//---------------------------------------------------------------------------------------------------------------
//
//  HAUD 2024.11.21
//
//
//  fb_Instance
//-----------------------------------------------------------------------------
//  - base class for my process instance to work with fb_ProcessCollector
//
//  - _nProcess --> whoami, this is me
//
//  - fb_ProcessCollector[_nProcess].Cycle() is called in APPLICATION(PRG)
//    - handles range of XtsStations
//    - range must be closed and in consecutive order
//
//    - combines states into bitmasks, one bit per XtsStation
//    - controls forwarding of commands to range of XtsStations 
//      (see fb_ProcessCollector.Cycle())
//
//  - reference to all _ItfProcessCollector(I_ProcessCollector)[]
//    - _ItfProcessCollector[nProcess] Get/Set properties and methods
//
//  - Control / State of my process
//    - datafield for control and state provided
//    - _Ctrl 
//      --> commands to my process; fb_ProcessCollector[_nProcess]
//      --> is linked (REF=) automatically in Check()
//
//      Cmd               : E_PROCESS_CTRL; // command enum for my process
//      ProcessTarget     : UINT;           // target of my process
//      ActivateStation   : WORD;           // is checked for every job
//                                          // every bit is a XtsStation
//
//      NestMask          : BYTE;           // one mask for all XtsStations
//      - every bit is a PosStop in a XtsStation
//      - copied to every XtsStation in my process when movers are about to leave
//
//    - _State
//      --> satus information from my process
//      --> check for plausible StationLast / StationFirst range of XtsStations
//
//      State             : E_PROCESS_STATE;  // state enuum from my process
//      Result            : E_PROGRESS;       // substate from my process, BUSY signals state is ready for interaction
//      Check             : E_PROCESS_CHECK;  // plausibility check of StationLast and StationFirst 
//
//
//  - basic check and var names, so you can build your procedures with it
//
//  - processes may be connected via linked list, you decide.
//    - linked list for processes is intended to work as job buffer
//    - linked list provides information via ST_PROCESS_DATA, 
//      add what you have to in there
//    - linked ist to all process instances provided
//
//  - inherit this base class for your application, call Check() cyclic
//
//---------------------------------------------------------------------------------------------------------------//
// This SOFTWARE is provided as an Example by THE PROVIDER "as is" and "with all faults." THE PROVIDER makes no  //
// representations or warranties of any kind concerning the safety, suitability, lack of viruses, inaccuracies,  //
// typographical errors, or other harmful components of this SOFTWARE. There are inherent dangers in the use of  //
// any software, and you are solely responsible for determining whether this SOFTWARE is compatible with your    //
// equipment and other software installed on your equipment. You are also solely responsible for the protection  //
// of your equipment and backup of your data, and THE PROVIDER will not be liable for any damages you may suffer //
// in connection with using, modifying, or distributing this SOFTWARE.                                           //
//---------------------------------------------------------------------------------------------------------------//
FUNCTION_BLOCK ABSTRACT fb_Instance
VAR
  // process index
  _nProcess               : E_INSTANCE;           // whoami

  _stInstanceCtrl         : REFERENCE TO ARRAY[1..MAX_PROCESS] OF ST_INSTANCE_CTRL;
  _stInstanceState        : REFERENCE TO ARRAY[1..MAX_PROCESS] OF ST_INSTANCE_STATE;

  _eCmd,
  _eCmdOld                : E_INSTANCE_CMD;       // commands for local state machine
  _eStateInstance         : E_INSTANCE_STATE;     // local state machine for infeed procedure

  _eResult,
  _eStateProgress         : E_PROGRESS;           // substate for lacal state machine

  _eInit                  : E_PROGRESS;           // startup
  _eCheck                 : E_INSTANCE_CHECK;     // pointer checks


  // local ctrl / state datafields for you to use, connected by reference to _ItfProcessCollector[_nProcess]
  _stCtrl                 : ST_PROCESS_CTRL;      // control to write, connected by reference to _ItfProcessCollector
  _stState                : ST_PROCESS_STATE;     // state   to read,  connected by reference to _ItfProcessCollector

  _ItfProcessCollector    : ARRAY[1..MAX_PROCESS] OF I_ProcessCollector;    // information and configuration of the connected ProcessCollector for given range of XtsStations

  _ItfProcessList         : ARRAY[1..MAX_PROCESS] OF I_Process_LinkedList;  // access to all linked lists for process entry
  _stListResult           : ST_PROCESS_LIST_RESULT;
  _stProcessData          : ST_PROCESS_DATA;

  {attribute 'displaymode':='bin'}
  _wTargetMask            : ARRAY[1..SIZEOF(T_PROCESS)*8] OF BYTE; // bits for PosStop[] to use in XtsStation of target process

  _stMsg                  : ST_Message;
  _MessageLevel           : E_MessageType;
END_VAR

METHOD Check : BOOL // call this method in the extending/inheriting class
//-----------------------------------------------------------------------------
//-----------------------------------------------------------------------------
// plausibility checks
//-----------------------------------------------------------------------------
IF NOT (_nProcess > 0)
THEN
  _eCheck                 := E_INSTANCE_CHECK.PROCESS_ID_ZERO;
  RETURN;
END_IF

IF NOT (_nProcess < E_INSTANCE.INSTANCE_MAX)
THEN
  _eCheck                 := E_INSTANCE_CHECK.PROCESS_ID_MAX;
  RETURN;
END_IF
//-----------------------------------------------------------------------------
//-----------------------------------------------------------------------------
// pointer checks
//-----------------------------------------------------------------------------
IF NOT __ISVALIDREF(_stInstanceCtrl)
THEN
  _eCheck                 := E_INSTANCE_CHECK.INVALID_INSTANCE_CONTROL_REFERENCE;
  RETURN;
END_IF

IF NOT __ISVALIDREF(_stInstanceState)
THEN
  _eCheck                 := E_INSTANCE_CHECK.INVALID_INSTANCE_STATE_REFERENCE;
  RETURN;
END_IF

IF NOT (_ItfProcessCollector[_nProcess] <> 0) 
THEN
  _eCheck                 := E_INSTANCE_CHECK.POINTER_COLLECTOR_ITF_INVALID;
  RETURN;
END_IF

IF NOT (_ItfProcessCollector[_nProcess].ProcessId > 0)
THEN
  _eCheck                 := E_INSTANCE_CHECK.PROCESS_ID_ZERO;
  RETURN;
END_IF

IF NOT (_ItfProcessCollector[_nProcess].ProcessId < E_INSTANCE.INSTANCE_MAX)
THEN
  _eCheck                 := E_INSTANCE_CHECK.PROCESS_ID_MAX;
  RETURN;
END_IF

IF NOT (_nProcess = _ItfProcessCollector[_nProcess].ProcessId)
THEN
  _eCheck                 := E_INSTANCE_CHECK.PROCESS_ID_NOTEQUAL_COLLECTOR_ID;
  RETURN;
END_IF

IF NOT (_ItfProcessList[_nProcess] <> 0)
THEN
  _eCheck                 := E_INSTANCE_CHECK.PROCESS_LIST_ITF_INDEX_INVALID;
  RETURN;
END_IF
//-----------------------------------------------------------------------------
//-----------------------------------------------------------------------------
// connect datafields to interface of ProcessCollector
//-----------------------------------------------------------------------------
_ItfProcessCollector[_nProcess].ProcessCtrl   REF= _stCtrl;
_ItfProcessCollector[_nProcess].ProcessState  REF= _stState;

//-----------------------------------------------------------------------------
//-----------------------------------------------------------------------------
// set message device
//-----------------------------------------------------------------------------
_stMsg.eDevice            := e_Device.Process + TO_UINT(_nProcess);
//-----------------------------------------------------------------------------
//-----------------------------------------------------------------------------
_eCheck                   := E_INSTANCE_CHECK.CHECK_DONE;
Check                     := TRUE;
END_METHOD

METHOD CmdLog

IF (_MessageLevel > E_MessageType.eMessageError)
THEN
  _stMsg.eSubdevice       := e_Subdevice.Instance_Command;
  _stMsg.iErrorNumber     := _nProcess;
  _stMsg.sText            := concat('E_INSTANCE_CMD', '.');
  _stMsg.sText            := concat(_stMsg.sText, TO_STRING(_eCmd));
  f_MessageSet(_stMsg);
END_IF
END_METHOD

PROPERTY CollectorInterface : array[1..MAX_PROCESS] of I_ProcessCollector
SET
_ItfProcessCollector := CollectorInterface;
END_SET
END_PROPERTY

PROPERTY InstanceCtrl : REFERENCE TO ARRAY[1..MAX_PROCESS] OF ST_INSTANCE_CTRL
SET
_stInstanceCtrl ref= InstanceCtrl;
END_SET
END_PROPERTY

PROPERTY InstanceState : REFERENCE TO ARRAY[1..MAX_PROCESS] OF ST_INSTANCE_STATE
SET
_stInstanceState ref= InstanceState;
END_SET
END_PROPERTY

PROPERTY MessageLevel : e_MessageType
GET
MessageLevel := _MessageLevel;
END_GET
SET
_MessageLevel := MessageLevel;

IF NOT (_eInit  = E_PROGRESS.PROGRESS_DONE) OR
   NOT (_eCheck = E_INSTANCE_CHECK.CHECK_DONE)
THEN
  RETURN;
ELSE
  _ItfProcessCollector[_nProcess].MessageLevel := _MessageLevel;
END_IF
END_SET
END_PROPERTY

PROPERTY ProcessId : E_INSTANCE
GET
ProcessId := _nProcess;
END_GET
SET
_nProcess := ProcessId;
END_SET
END_PROPERTY

PROPERTY ProcessLinkedLists : ARRAY[1..max_process] OF I_Process_LinkedList
SET
_ItfProcessList := ProcessLinkedLists;
END_SET
END_PROPERTY

END_FUNCTION_BLOCK

(* stored: Version 1.1.0.1
   POU fb_Instance: Id {9ff3c516-45ba-4b78-9d4b-75122957572f}, SpecialFunc None
   Folder properties: Id {d004a5e1-40ce-456b-9e1d-ee64800d3a3e}
   Method Check: Id {26e2c889-643e-4b01-93d5-649397b5681a}
   Method CmdLog: Id {718a7c87-90df-41eb-b260-c94b8c7d6a49}
   Property CollectorInterface: Id {cfcc05b8-33ec-47e0-8abd-f04ff243a3e1}
   Set Set: Id {68af5d0f-0bf0-45fe-bb34-1ce8589a81a7}
   Property InstanceCtrl: Id {6ab36380-0aaa-4815-9ffb-43233cec73c7}
   Set Set: Id {014e092e-2708-41bb-b142-069575403ce2}
   Property InstanceState: Id {2c28eb5f-87bc-4dab-b067-d0c20b147b79}
   Set Set: Id {8fe48b09-9a26-41d0-bc7d-cb0ed1bb80bd}
   Property MessageLevel: Id {5a2196b9-a9df-488d-bdb8-e4cf3ce67041}
   Get Get: Id {8e32f2a1-13b9-4567-98d3-a86088a15e12}
   Set Set: Id {e1d47b21-3a6c-4308-9376-d5ddc069753f}
   Property ProcessId: Id {3a74a077-94e7-4198-956c-bad99d4e7d74}
   Get Get: Id {4e0e1cf7-73ea-4d73-a2e9-0e3380160835}
   Set Set: Id {00dbfc55-d45d-4e86-8382-97a98599211f}
   Property ProcessLinkedLists: Id {e443e036-df37-43bb-a5af-39e86753633f}
   Set Set: Id {2ece14d1-28f1-4e19-9aac-76d96b236cb0} *)
